Staubli VAL3: changePCircle.pgx

public program changePCircle(num x_nIndex)
  local bool l_bOk
  local bool l_bRefresh
  local bool l_bUnreach
  local frame l_fTraj
  local joint l_jJoint
  local num l_nIndex
  local num l_nKey
  local num l_nMoveId
  local num l_nResult[2]
  local num l_nView
  local point l_pPoint[2]
  local string l_sButton[2]
  local string l_sEvent
  local string l_sItem
  local string l_sMessage
  local tool l_tTool
  local trsf l_tTrsf
  local trsf l_tTrsfTemp[2]
  local trsf l_trsfPoint
begin
  // INIT
  l_bRefresh=false
  l_nIndex=0
  l_nView=0
  call use:setSizeList(10,3,20,6)
  call use:setView(false)
  // get the tool
  call tcp:getTool(l_tTool,pEditPoint.nIndexTool)
  // get the point and the circle point
  call getPoint(l_pPoint,false,x_nIndex)
  // point final
  pPoints=l_pPoint
  // point intermediare
  pPoints[1]=l_pPoint[1]
  l_tTrsf=l_pPoint[1].trsf
  //
  do
    // check if the intermediate point is reachable
    call isReachable(l_pPoint[1],l_tTool,l_bUnreach)
    //move to
    if cycleStatus:nWorkingMode==1 and !cycleStatus:bCycle and !cycleStatus:bSimulation and !l_bUnreach
      // empty the stack
      resetMotion()
      if distance(here(l_tTool,pEditPoint.fFrame),pPoints[1])>1
        call checkPCircle(x_nIndex,here(l_tTool,pEditPoint.fFrame),l_nResult)
        // CIRCULAR MOVE
        if l_nResult!=-1
          // find P.I. percentage
          call checkPCircle(x_nIndex,pPoints[1],l_nResult[1])
          // take the previous point
          call getPoint(l_pPoint,false,x_nIndex-1)
          //
          // find the intermediate point
          //
          l_pPoint[1]=pPoints[1]
          pPoints[1].trsf=interpolateC(l_pPoint.trsf,pPoints[1].trsf,pPoints.trsf,(l_nResult+l_nResult[1])/2)
          // go to the intermediate point
          pPoints[0]=l_pPoint[1]
          movec(pPoints[1],pPoints,l_tTool,mMdesc)
        else
          // joint MOVE
          movej(pPoints[1],l_tTool,mMdesc)
        endIf
        // joint MOVE
      else
        // joint MOVE
        movej(pPoints[1],l_tTool,mMdesc)
      endIf
    endIf
    // show the menu
    call use:clear(0,13)
    call use:typeMenu(8,"OK")
    if !cycleStatus:bCycle and !cycleStatus:bSimulation
      call use:typeMenu(1,"Here")
    endIf
    // show the context
    call use:listcreate("")
    l_sMessage="coord  X > "+toString(".2",l_tTrsf.x)
    call use:listadd(l_sMessage)
    l_sMessage="coord  Y > "+toString(".2",l_tTrsf.y)
    call use:listadd(l_sMessage)
    l_sMessage="coord  Z > "+toString(".2",l_tTrsf.z)
    call use:listadd(l_sMessage)
    l_sMessage="coord RX > "+toString(".2",l_tTrsf.rx)
    call use:listadd(l_sMessage)
    l_sMessage="coord RY > "+toString(".2",l_tTrsf.ry)
    call use:listadd(l_sMessage)
    l_sMessage="coord RZ > "+toString(".2",l_tTrsf.rz)
    call use:listadd(l_sMessage)
    use:nView=l_nIndex
    call use:listupdate(l_nIndex-l_nView)
    // edit the items
    do
      l_nView=use:nView
      l_nKey=get()
      call use:listevent(l_nKey,l_nIndex,l_sEvent)
      switch l_nKey
        case 271
          // here POINT
          if !cycleStatus:bCycle and !cycleStatus:bSimulation
            // ASK IF YOU WANT TO RECORD THE POINT
            call language:message(l_sMessage,131)
            call language:getYesNo(l_sButton)
            call use:yes_no(l_sMessage,l_sButton,l_bOk)
            if l_bOk
              call HerePointCircle(x_nIndex)
            endIf
          endIf
        break
        case 270
          // clean the line
          call use:listcursor(use:nView,false)
          // EDIT FIELD
          switch l_nIndex
            case 0
              //  x-value
              l_sItem=""
              call use:changeValue(l_tTrsf.x,0,0,2+40-use:nBottomX,use:nView+1+3,l_sItem)
            break
            case 1
              //  y-value
              l_sItem=""
              call use:changeValue(l_tTrsf.y,0,0,2+40-use:nBottomX,use:nView+1+3,l_sItem)
            break
            case 2
              //  z-value
              l_sItem=""
              call use:changeValue(l_tTrsf.z,0,0,2+40-use:nBottomX,use:nView+1+3,l_sItem)
            break
            case 3
              //  rx-value
              l_sItem=""
              call use:changeValue(l_tTrsf.rx,0,0,2+40-use:nBottomX,use:nView+1+3,l_sItem)
            break
            case 4
              //  ry-value
              l_sItem=""
              call use:changeValue(l_tTrsf.ry,0,0,2+40-use:nBottomX,use:nView+1+3,l_sItem)
            break
            case 5
              //  rz-value
              l_sItem=""
              call use:changeValue(l_tTrsf.rz,0,0,2+40-use:nBottomX,use:nView+1+3,l_sItem)
            break
          endSwitch
          l_bRefresh=true
        break
      endSwitch
      delay(0)
    until l_bRefresh==true or l_nKey==255 or l_nKey==278 or l_nKey==271
    //
    // check if is OK   VALUE CHANGE
    //
    if l_nKey==270
      pPoints[1].trsf=l_pPoint[1].trsf=l_tTrsf
    endIf
    //
    l_bRefresh=false
    delay(0)
  until l_nKey==255 or l_nKey==278 or l_nKey==271 or l_bUnreach
  //
  // save the data
  //
  if l_nKey==278
    // record it
    if !l_bUnreach
      // update the circle point
      pEditPoint.tData[x_nIndex].pCircle.trsf=l_tTrsf
    endIf
  endIf
  // release the resource
  call use:nullKey(l_nKey)
end
